TYPE Uc_List :
STRUCT
	nSelected			: UINT;
	ptSelected			: POINTER TO BYTE;
	astEntries			: ARRAY[0..255] OF ST_Listentry;
	bRemove				: BOOL;
	bInsert				: BOOL;
	bMoveUp				: BOOL;
	bMoveDown			: BOOL;
	bSave				: BOOL;
END_STRUCT
END_TYPE

(* stored: Version 1.1.0.1
   DUT Uc_List: Id {a68e73ea-f608-4f4e-bbf3-02fa139a30ac} *)
